// TIA Portal V20 export
FUNCTION_BLOCK "Simulation"   // FB32838, LAD
// stored: MemoryReserve 100, Namespace Unit1.Em6, SetENOAutomatically false
   VAR_INPUT
      simulation { ExternalAccessible := 'False'; ExternalVisible := 'False'; ExternalWritable := 'False'} : Bool;
   END_VAR
   VAR
      instActuator { ExternalAccessible := 'False'; ExternalVisible := 'False'; ExternalWritable := 'False'} : Array[0..9] of "Simulation_Actuator";
      statDigitalSignal { ExternalAccessible := 'False'; ExternalVisible := 'False'; ExternalWritable := 'False'} : Array[0..9] of Bool;
   END_VAR
   VAR_TEMP   // added for the SCL form of the ladder/FBD networks
      _w1 : Bool;
   END_VAR
BEGIN

REGION Network 1: Digital Signal
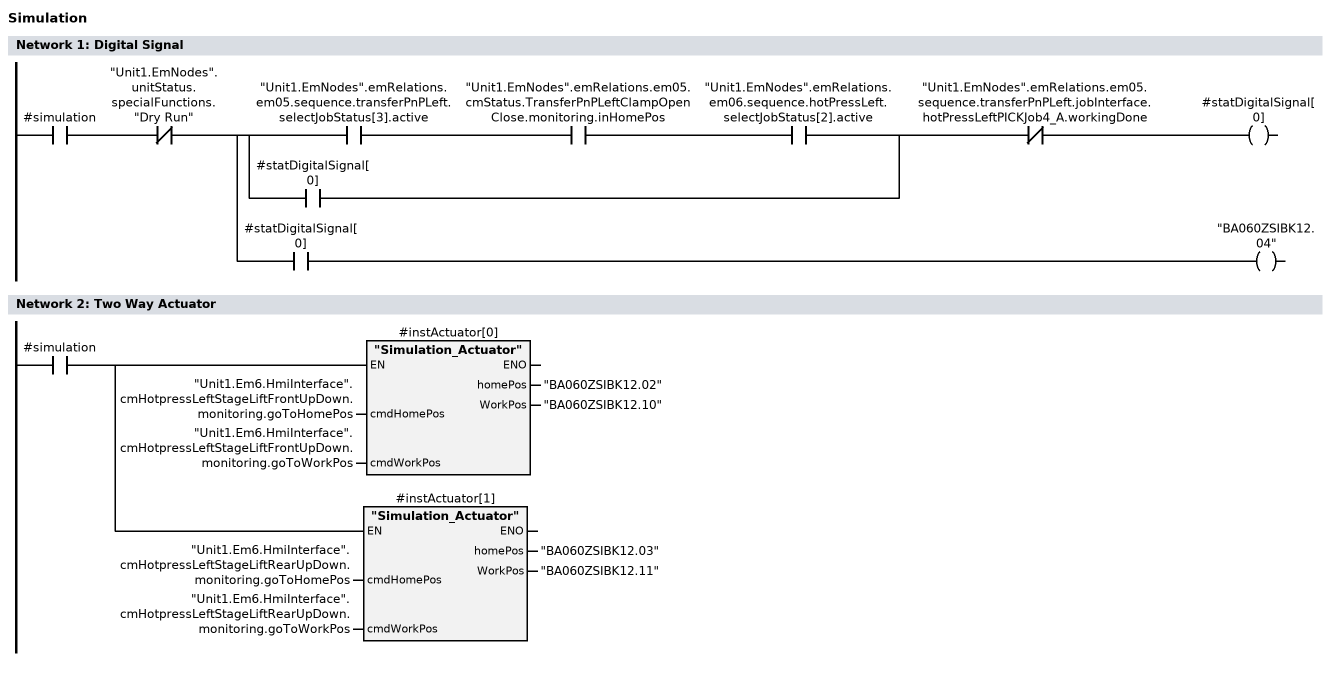
   RUNG wire#powerrail
      Contact( #simulation )
      I_Contact( "Unit1.EmNodes".unitStatus.specialFunctions."Dry Run" )
      wire#w1
      Contact( "Unit1.EmNodes".emRelations.em05.sequence.transferPnPLeft.selectJobStatus[3].active )
      Contact( "Unit1.EmNodes".emRelations.em05.cmStatus.TransferPnPLeftClampOpenClose.monitoring.inHomePos )
      Contact( "Unit1.EmNodes".emRelations.em06.sequence.hotPressLeft.selectJobStatus[2].active )
      wire#w2
      I_Contact( "Unit1.EmNodes".emRelations.em05.sequence.transferPnPLeft.jobInterface.hotPressLeftPICKJob4_A.workingDone )
      Coil( #statDigitalSignal[0] )
   END_RUNG
   RUNG wire#w1
      Contact( #statDigitalSignal[0] )
   END_RUNG wire#w2
   RUNG wire#w1
      Contact( #statDigitalSignal[0] )
      Coil( "BA060ZSIBK12.04" )
   END_RUNG
   // the same network as SCL:
   #_w1 := #simulation AND NOT "Unit1.EmNodes".unitStatus.specialFunctions."Dry Run";
   #statDigitalSignal[0] := #_w1 AND (("Unit1.EmNodes".emRelations.em05.sequence.transferPnPLeft.selectJobStatus[3].active AND "Unit1.EmNodes".emRelations.em05.cmStatus.TransferPnPLeftClampOpenClose.monitoring.inHomePos AND "Unit1.EmNodes".emRelations.em06.sequence.hotPressLeft.selectJobStatus[2].active) OR #statDigitalSignal[0]) AND NOT "Unit1.EmNodes".emRelations.em05.sequence.transferPnPLeft.jobInterface.hotPressLeftPICKJob4_A.workingDone;
   "BA060ZSIBK12.04" := #_w1 AND #statDigitalSignal[0];
END_REGION

REGION Network 2: Two Way Actuator
   RUNG wire#powerrail
      Contact( #simulation )
      wire#w1
      #instActuator[0](cmdHomePos := "Unit1.Em6.HmiInterface".cmHotpressLeftStageLiftFrontUpDown.monitoring.goToHomePos, cmdWorkPos := "Unit1.Em6.HmiInterface".cmHotpressLeftStageLiftFrontUpDown.monitoring.goToWorkPos, homePos => "BA060ZSIBK12.02", WorkPos => "BA060ZSIBK12.10")
   END_RUNG
   RUNG wire#w1
      #instActuator[1](cmdHomePos := "Unit1.Em6.HmiInterface".cmHotpressLeftStageLiftRearUpDown.monitoring.goToHomePos, cmdWorkPos := "Unit1.Em6.HmiInterface".cmHotpressLeftStageLiftRearUpDown.monitoring.goToWorkPos, homePos => "BA060ZSIBK12.03", WorkPos => "BA060ZSIBK12.11")
   END_RUNG
   // the same network as SCL:
   IF #simulation THEN
       #instActuator[0](cmdHomePos := "Unit1.Em6.HmiInterface".cmHotpressLeftStageLiftFrontUpDown.monitoring.goToHomePos,   // "Simulation_Actuator"
                        cmdWorkPos := "Unit1.Em6.HmiInterface".cmHotpressLeftStageLiftFrontUpDown.monitoring.goToWorkPos,
                        homePos => "BA060ZSIBK12.02",
                        WorkPos => "BA060ZSIBK12.10");
       #instActuator[1](cmdHomePos := "Unit1.Em6.HmiInterface".cmHotpressLeftStageLiftRearUpDown.monitoring.goToHomePos,   // "Simulation_Actuator"
                        cmdWorkPos := "Unit1.Em6.HmiInterface".cmHotpressLeftStageLiftRearUpDown.monitoring.goToWorkPos,
                        homePos => "BA060ZSIBK12.03",
                        WorkPos => "BA060ZSIBK12.11");
   END_IF;
END_REGION
END_FUNCTION_BLOCK
